// TIA Portal V18 export
PlcTagTable "Default tag table"
  PlcTag "HMI_Run_Enable"  LogicalAddress=%M20.0
  PlcTag "HMI_Reset_Alarm"  LogicalAddress=%M20.1
  PlcTag "HMI_Sim_Mode"  LogicalAddress=%M20.2
  PlcTag "PLC2_State"  LogicalAddress=%MW12
  PlcTag "PLC2_Loi_Tong"  LogicalAddress=%M20.3
  PlcTag "PLC2_Stop_Active"  LogicalAddress=%M20.4
  PlcTag "PLC2_EStop_Latch"  LogicalAddress=%M20.5
  PlcTag "PID_Bon4_Enable"  LogicalAddress=%M20.6
  PlcTag "PID_Bon4_SP"  LogicalAddress=%MD30
  PlcTag "PID_Bon4_PV"  LogicalAddress=%MD34
  PlcTag "PID_Bon4_CV"  LogicalAddress=%MD38
  PlcTag "HMI_SP_PLC2_Nhiet_Do_Bon4"  LogicalAddress=%MD42
  PlcTag "TT3219_Bon4_Sim"  LogicalAddress=%MD46
  PlcTag "CV3216_Hoi_Bon4"  LogicalAddress=%MD50
  PlcTag "MB_TCP_Server_Error"  LogicalAddress=%M20.7
  PlcTag "MB_TCP_Server_Busy"  LogicalAddress=%M21.0
  PlcTag "MB_TCP_Server_NDR"  LogicalAddress=%M21.1
  PlcTag "MB_TCP_Server_DR"  LogicalAddress=%M21.2
  PlcTag "PLC2_Heartbeat_Timeout"  LogicalAddress=%M21.3
  PlcTag "MB_TCP_Server_Status"  LogicalAddress=%MW54
  PlcTag "PLC2_Heartbeat"  LogicalAddress=%MW56
  PlcTag "PLC1_Heartbeat_Recv"  LogicalAddress=%MW58
  PlcTag "CV3211_Nuoc_Bon3_M"  LogicalAddress=%MD1216
  PlcTag "CV3216_Hoi_Bon4_M"  LogicalAddress=%MD1224
  PlcTag "FQ3210_Bon3_Eff"  LogicalAddress=%MD776
  PlcTag "FQ3215_Bon4_Eff"  LogicalAddress=%MD808
  PlcTag "HMI_Anim_Bon3_Frame"  LogicalAddress=%MW260
  PlcTag "HMI_Anim_Bon3_MucDich"  LogicalAddress=%MW262
  PlcTag "HMI_Anim_Bon4_Frame"  LogicalAddress=%MW264
  PlcTag "HMI_Anim_Bon4_MucDich"  LogicalAddress=%MW266
  PlcTag "LT3213_Bon3_Eff"  LogicalAddress=%MD784
  PlcTag "LT3218_Bon4_Eff"  LogicalAddress=%MD816
  PlcTag "TT3214_Bon3_Eff"  LogicalAddress=%MD792
  PlcTag "TT3219_Bon4_Eff"  LogicalAddress=%MD824
  PlcTag "V3240_Nuoc_Bon3"  LogicalAddress=%M100.0
  PlcTag "V3242_Xa_Bon3"  LogicalAddress=%M100.1
  PlcTag "V3243_Xa_Bon3"  LogicalAddress=%M100.2
  PlcTag "V3244_Xa_Bon3"  LogicalAddress=%M100.3
  PlcTag "V3245_Nuoc_Bon4"  LogicalAddress=%M100.4
  PlcTag "V3247_Xa_Bon4"  LogicalAddress=%M100.5
  PlcTag "V3248_Xa_Bon4"  LogicalAddress=%M100.6
  PlcTag "V3249_Xa_Bon4"  LogicalAddress=%M100.7
  PlcTag "HMI_SP_PLC2_Nuoc_Bon3"  LogicalAddress=%MD916
  PlcTag "HMI_SP_PLC2_Nuoc_Bon4"  LogicalAddress=%MD920
  PlcTag "HMI_SP_Time_Khuay_Bon3"  LogicalAddress=%MD948
